TYPE ST_CartInfo :
STRUCT
	//joint position-unit:rad/m
	m_curJntPos:Vec8d;
	
	//joint position-unit:deg/mm
	m_curJntPosDegMM:Vec8d;
	
	//current joint velocity
	m_curJntVelDegMM:Vec8d;
	
	//link position
	m_curLinkPos:Vec8d;
	
	//Encoder deviation
	m_encErr:Vec8d;
	
	//joint maxmum
	m_jntMax:Vec8d;
	
	//joint minimum
	m_jntMin:Vec8d;
	
	//motor input signal
	m_motorInput:ARRAY[1..8] OF ST_MotorInputs;
	
	//motor output signal
	m_motorOutput:ARRAY[1..8] OF ST_MotorOutputs;
	
	//state machine
	m_stateMachine:INT;
	
	//IP Address
	m_IPAddress:T_AmsNetId;
END_STRUCT
END_TYPE

(* stored: Version 1.1.0.1, ProductVersion 3.1.4024.11
   DUT ST_CartInfo: Id {d60cba0c-b85c-42ee-843d-a5ac9829e21c} *)
